// TwinCAT 3 PLC project MotionControl
// ProgramVersion: 3.1.4022.6
// libraries:
//   Tc2_MC2, * (Beckhoff Automation GmbH)
//   Tc2_Standard, * (Beckhoff Automation GmbH)
//   Tc2_System, * (Beckhoff Automation GmbH)
//   Tc3_Module, * (Beckhoff Automation GmbH)
//   Tc3_mxAutomation, * (Beckhoff Automation GmbH)
//   Tc3_mxAutomationV3_0, * (Beckhoff Automation GmbH)
//   Tc3_uniValPlc, * (Beckhoff Automation GmbH)
// project tree:
//   / GlobalTextList.TcGTLO, PlcTask.TcTTO, Visualization Manager.TcVMO (not stored)
//   POUs/ MAIN.TcPOU
//   VISUs/ Visualization.TcVIS
// real-time tasks:
//   TASK PlcTask: cycle T#10ms, priority 20, ADS port 350
// motion (NC):
//   TASK NC-Task 1 SAF: cycle T#2ms, priority 4, ADS port 501
//   TASK NC-Task 1 SVB: cycle T#10ms, priority 8, ADS port 511
//   AXIS ACS1 (id 1)
//     OtherSettings: AllowMotionCmdToSlave=true
//     encoder EncType=1
//     drive DrvType=5
//       Analog: ScaleFactorActTorque=0.1
//       TimeComp: TaskDelayCycles=1
//     controller CtrType=1
//       CtrPara: PriorControlFactor=1
//         Observer: BandWidth=20
//   AXIS ACS2 (id 2)
//     OtherSettings: AllowMotionCmdToSlave=true
//     encoder EncType=1
//     drive DrvType=5
//       Analog: ScaleFactorActTorque=0.1
//       TimeComp: TaskDelayCycles=1
//     controller CtrType=1
//       CtrPara: PriorControlFactor=1
//         Observer: BandWidth=20
//   AXIS ACS3 (id 3)
//     OtherSettings: AllowMotionCmdToSlave=true
//     encoder EncType=1
//     drive DrvType=5
//       Analog: ScaleFactorActTorque=0.1
//       TimeComp: TaskDelayCycles=1
//     controller CtrType=1
//       CtrPara: PriorControlFactor=1
//         Observer: BandWidth=20
//   AXIS MCS1 (id 4)
//     OtherSettings: AllowMotionCmdToSlave=true
//     encoder EncType=1
//     drive DrvType=5
//       Analog: ScaleFactorActTorque=0.1
//       TimeComp: TaskDelayCycles=1
//     controller CtrType=1
//       CtrPara: PriorControlFactor=1
//         Observer: BandWidth=20
//   AXIS MCS2 (id 5)
//     OtherSettings: AllowMotionCmdToSlave=true
//     encoder EncType=1
//     drive DrvType=5
//       Analog: ScaleFactorActTorque=0.1
//       TimeComp: TaskDelayCycles=1
//     controller CtrType=1
//       CtrPara: PriorControlFactor=1
//         Observer: BandWidth=20
//   AXIS MCS3 (id 6)
//     OtherSettings: AllowMotionCmdToSlave=true
//     encoder EncType=1
//     drive DrvType=5
//       Analog: ScaleFactorActTorque=0.1
//       TimeComp: TaskDelayCycles=1
//     controller CtrType=1
//       CtrPara: PriorControlFactor=1
//         Observer: BandWidth=20
// variable links:
//   MotionControl/MotionControl Instance <-> NC-Task 1 SAF/Axes/ACS1
//     PlcTask Inputs/MAIN.masterAxis.NcToPlc <-> Outputs/ToPlc
//     PlcTask Outputs/MAIN.masterAxis.PlcToNc <-> Inputs/FromPlc
//   MotionControl/MotionControl Instance <-> NC-Task 1 SAF/Axes/ACS2
//     PlcTask Inputs/MAIN.slaveAxis.NcToPlc <-> Outputs/ToPlc
//     PlcTask Outputs/MAIN.slaveAxis.PlcToNc <-> Inputs/FromPlc
//   MotionControl/MotionControl Instance <-> NC-Task 1 SAF/Channel 2
//     PlcTask Inputs/MAIN.in_stKinToPlc <-> Outputs/ToPlc
//     PlcTask Outputs/MAIN.out_stPlcToKin <-> Inputs/FromPlc

CONFIGURATION MotionControl
    RESOURCE PLC ON TwinCAT3
        TASK PlcTask(INTERVAL := T#10ms, PRIORITY := 20);
        PROGRAM MAIN WITH PlcTask : MAIN;
    END_RESOURCE
END_CONFIGURATION

// ---- POUs/MAIN.TcPOU
PROGRAM MAIN
VAR
	masterAxis : Axis_Ref;
	slaveAxis  : Axis_Ref;
	
	fb_masterStatus : MC_ReadStatus;
	fb_slaveStatus 	: MC_ReadStatus;
	
	fb_masterPower :MC_Power;
	fb_slavePower : MC_Power;
	
	fb_synchronize :MC_GearIn;
	
	fb_moveRelative : MC_MoveRelative;

	
	state		: INT;
	bPower		: BOOL;
	bMove		: BOOL;
	nDistance	: LREAL := 500;
	nVelocity	: LREAL := 50;
END_VAR


CASE state OF
	0: 	//Idle case
	
	fb_masterStatus(
		Axis := masterAxis,
		Enable := TRUE);
		
	fb_slaveStatus(
		Axis := slaveAxis,
		Enable := TRUE);
		
	IF NOT fb_masterStatus.Error AND NOT fb_slaveStatus.Error THEN
		state := 10;
	END_IF
	
	10: 	//Power up motors
	
	IF NOT fb_masterPower.Status THEN
		fb_masterPower.Enable := NOT bPower;
	END_IF
	
	fb_masterPower(
		Axis := masterAxis,
		Enable := bPower,
		Enable_Positive := bPower,
		Enable_Negative := bPower);
		
	fb_slavePower(
		Axis := slaveAxis,
		Enable := bPower,
		Enable_Positive := bPower,
		Enable_Negative := bPower);		
	
	IF fb_masterPower.Status AND fb_slavePower.Status THEN
		state := 20;
	END_IF
	
	20: 	//Synchronize motors
	IF NOT fb_synchronize.InGear THEN
		fb_synchronize.Execute := FALSE;
	END_IF
	
	fb_synchronize(
		Master := masterAxis,
		Slave := slaveAxis,
		Execute := TRUE);
		
	IF fb_synchronize.InGear THEN
		state := 30;
	END_IF

	30: 	//Move relative 500mm at 50mm/s
	
	fb_moveRelative(
		Axis := masterAxis,
		Execute := bMove,
		Distance := nDistance,
		Velocity := nVelocity);
END_CASE

END_PROGRAM

// ---- GlobalTextList.TcGTLO
TEXTLIST GlobalTextList
  878 = 'Error status'
  275 = 'Master'
  738 = 'Slave'
END_TEXTLIST

// ---- VISUs/Visualization.TcVIS
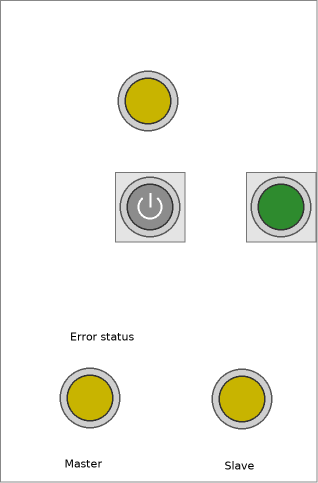
VISUALIZATION Visualization  // 318x483
    Lamp1 (113,66 70x70), variable: MAIN.fb_masterPower.Status, style: Lamp-Lamp1-Yellow
    PowerSwitch (115,172 70x70), variable: MAIN.bPower, behaviour: TOGGLE, style: Switch-PowerSwitch-Gray
    Lamp1 (55,363 70x70), variable: MAIN.fb_masterStatus.Error, style: Lamp-Lamp1-Yellow
    Lamp1 (207,364 70x70), variable: MAIN.fb_slaveStatus.Error, style: Lamp-Lamp1-Yellow
    Label (39,449 89x30), "Master"
    Label (197,451 85x30), "Slave"
    Label (54,322 96x30), "Error status"
    PushSwitch (246,172 70x70), variable: MAIN.bMove, behaviour: TAP, style: Switch-PushSwitch-Green
END_VISUALIZATION
